(* Logix 5000 project; controller Boca_de_Pescado Emulate 5570 rev 30.12; software revision 30.00 *)

TASK MainTask (continuous, watchdog 500 ms) : MainProgram

MODULES
   Local : Emulate 5570 (ICP 2, rev 30.12)
      VIRTUAL_OUTPUTS : vendor 1 type 0 code 15 (ICP 4, rev 1.1, Output RPI 50 ms)
      VIRTUAL_INPUTS : vendor 1 type 0 code 15 (ICP 3, rev 1.1, Output RPI 50 ms)
END_MODULES

PROGRAM MainProgram   (* main routine MainRoutine *)
VAR
   Action_000 : SFC_ACTION := (Status := 16#0020_0000, PauseTimer := 1);
   Action_001 : SFC_ACTION := (Status := 16#0020_0000, PauseTimer := 1);
   Action_002 : SFC_ACTION := (Status := 16#0020_0000, PauseTimer := 1);
   Action_003 : SFC_ACTION := (Status := 16#0020_0000, PauseTimer := 1);
   Action_004 : SFC_ACTION := (Status := 16#0020_0000, PauseTimer := 1);
   Action_005 : SFC_ACTION := (Status := 16#0020_0000, PauseTimer := 1);
   Action_006 : SFC_ACTION := (Status := 16#0020_0000, PauseTimer := 1);
   Action_007 : SFC_ACTION := (Status := 16#0020_0000, PauseTimer := 1);
   Action_008 : SFC_ACTION := (Status := 16#0020_0000, PauseTimer := 1);
   Action_009 : SFC_ACTION := (Status := 16#0020_0000, PauseTimer := 1);
   Action_010 : SFC_ACTION := (Status := 16#0020_0000, PauseTimer := 1);
   Action_011 : SFC_ACTION := (Status := 16#0020_0000, PauseTimer := 1);
   Action_012 : SFC_ACTION := (Status := 16#0020_0000, PauseTimer := 1);
   Counter : INT;
   H1 : BOOL;
   H2 : BOOL;
   H3 : BOOL;
   RST : BOOL;
   S1 : BOOL;
   S2 : BOOL;
   S3 : BOOL;
   S4 : BOOL;
   S5 : BOOL;
   S6 : BOOL;
   S7 : BOOL;
   START : BOOL;
   Step_00 : SFC_STEP := (Status := 16#0020_0000, PauseTimer := 1);
   Step_000 : SFC_STEP := (Status := 16#0020_0000, PauseTimer := 1);
   Step_001 : SFC_STEP := (Status := 16#0020_0000, PauseTimer := 1);
   Step_002 : SFC_STEP := (Status := 16#0020_0000, PauseTimer := 1, PRE := 1000);
   Step_003 : SFC_STEP := (Status := 16#0020_0000, PauseTimer := 1);
   Step_004 : SFC_STEP := (Status := 16#0020_0000, PauseTimer := 1);
   Step_005 : SFC_STEP := (Status := 16#0020_0000, PauseTimer := 1);
   Step_006 : SFC_STEP := (Status := 16#0020_0000, PauseTimer := 1);
   Step_007 : SFC_STEP := (Status := 16#0020_0000, PauseTimer := 1);
   Step_008 : SFC_STEP := (Status := 16#0020_0000, PauseTimer := 1);
   Step_009 : SFC_STEP := (Status := 16#0020_0000, PauseTimer := 1);
   Step_010 : SFC_STEP := (Status := 16#0020_0000, PauseTimer := 1);
   STOP_ALARM : BOOL;
   Tran_000 : BOOL;
   Tran_001 : BOOL;
   Tran_002 : BOOL;
   Tran_003 : BOOL;
   Tran_004 : BOOL;
   Tran_005 : BOOL;
   Tran_006 : BOOL;
   Tran_007 : BOOL;
   Tran_008 : BOOL;
   Tran_009 : BOOL;
   Tran_010 : BOOL;
   Tran_011 : BOOL;
   Tran_012 : BOOL;
   Tran_013 : BOOL;
   Y1 : BOOL;
   Y2 : BOOL;
   Y3 : BOOL;
   Y4 : BOOL;
   Y5 : BOOL;
   Y6 : BOOL;
END_VAR

ROUTINE MainRoutine   (* ladder *)
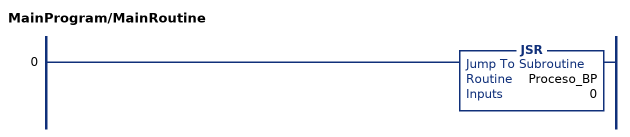
   0: JSR(Proceso_BP,0);
END_ROUTINE

ROUTINE Proceso_BP   (* sequential function chart *)
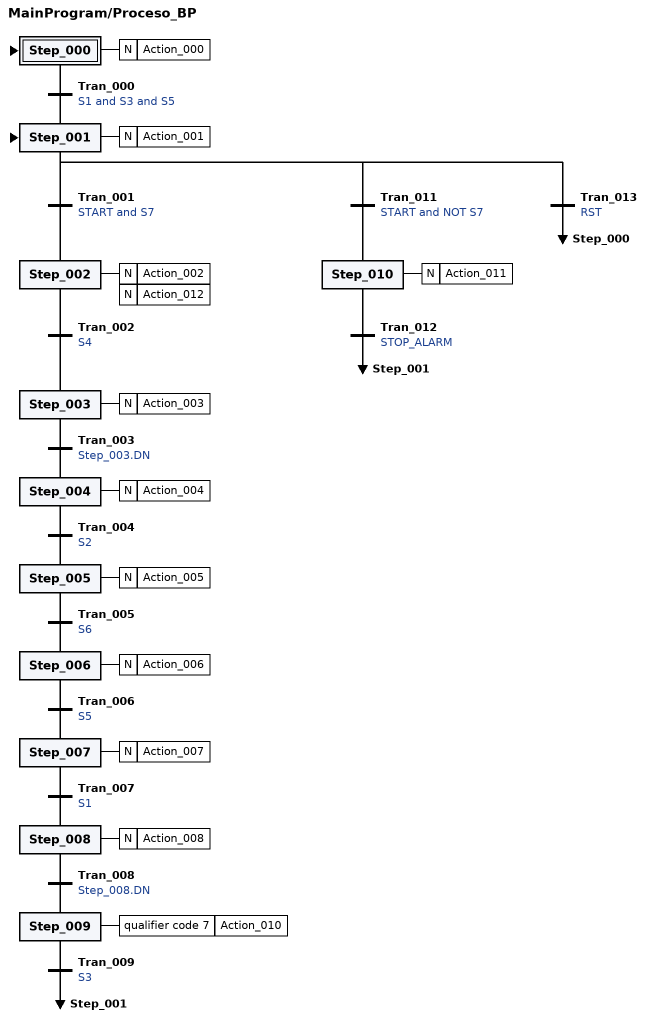
   INITIAL_STEP Step_000:
      ACTION Action_000 (N):
         Y1:=0;
         Y2:=1;
         Y3:=0;
         Y4:=1;
         Y5:=0;
         Y6:=1;
         H1:=0;
         H2:=0;
         H3:=0;
         Counter:=0;
         
         
      END_ACTION
   END_STEP
   TRANSITION Tran_000 FROM Step_000 TO Step_001
      := S1 and S3 and S5
         
   END_TRANSITION
   STEP Step_001:
      ACTION Action_001 (N):
         H1:=1;
         H2:=0;
         H3:=0;
         Y2:=0;
         Y4:=0;
         Y6:=0;
      END_ACTION
   END_STEP
   TRANSITION Tran_001 FROM Step_001 TO Step_002
      := START and S7
   END_TRANSITION
   TRANSITION Tran_011 FROM Step_001 TO Step_010
      := START and NOT S7
   END_TRANSITION
   TRANSITION Tran_013 FROM Step_001 TO Step_000
      := RST
   END_TRANSITION
   STEP Step_002:
      ACTION Action_002 (N):
         Y3:=1;
         Y4:=0;
      END_ACTION
      ACTION Action_012 (N):
         H2:=1;
         H1:=0;
      END_ACTION
   END_STEP
   STEP Step_010:
      ACTION Action_011 (N):
         H3:=1;
         H2:=0;
         H1:=0;
      END_ACTION
   END_STEP
   TRANSITION Tran_012 FROM Step_010 TO Step_001
      := STOP_ALARM
   END_TRANSITION
   TRANSITION Tran_002 FROM Step_002 TO Step_003
      := S4
   END_TRANSITION
   STEP Step_003:
      ACTION Action_003 (N):
         Y3:=0;
      END_ACTION
   END_STEP
   TRANSITION Tran_003 FROM Step_003 TO Step_004
      := Step_003.DN
   END_TRANSITION
   STEP Step_004:
      ACTION Action_004 (N):
         Y1:=1;
         
      END_ACTION
   END_STEP
   TRANSITION Tran_004 FROM Step_004 TO Step_005
      := S2
   END_TRANSITION
   STEP Step_005:
      ACTION Action_005 (N):
         Y5:=1;
         Y1:=0;
      END_ACTION
   END_STEP
   TRANSITION Tran_005 FROM Step_005 TO Step_006
      := S6
   END_TRANSITION
   STEP Step_006:
      ACTION Action_006 (N):
         Y6:=1;
         Y5:=0;
      END_ACTION
   END_STEP
   TRANSITION Tran_006 FROM Step_006 TO Step_007
      := S5
   END_TRANSITION
   STEP Step_007:
      ACTION Action_007 (N):
         Y2:=1;
         Y6:=0;
      END_ACTION
   END_STEP
   TRANSITION Tran_007 FROM Step_007 TO Step_008
      := S1
   END_TRANSITION
   STEP Step_008:
      ACTION Action_008 (N):
         Y4:=1;
         Y2:=0;
      END_ACTION
   END_STEP
   TRANSITION Tran_008 FROM Step_008 TO Step_009
      := Step_008.DN
   END_TRANSITION
   STEP Step_009:
      ACTION Action_010 (qualifier code 7):
         Counter:=Counter+1;
      END_ACTION
   END_STEP
   TRANSITION Tran_009 FROM Step_009 TO Step_001
      := S3
   END_TRANSITION
END_ROUTINE
END_PROGRAM
